{attribute 'GeneratedUsingTerminal: EK1122-0000-0018'}
{attribute addProperty BoxType "EK1122-0000-0018"}
{attribute addProperty Id "R1_A4_X2_A2_VI1_AES_D_BC_ECAT_xAES_B47A261080REX_350_IMecat_xIMecat_x_75C6CB6B170"}
{attribute addProperty CRC "967560231"}
{attribute addProperty Size "250"}
{attribute addProperty Name "R1_A4_X2_A2 (EK1122)"}
TYPE R1_A4_X2_A2_EK1122_39ABCC27 EXTENDS EK1122_1FC0878B :
STRUCT
	{attribute addProperty Name "R1_A4_X2_A2_VI1 (AES-D-BC-ECAT)"}
	{attribute addProperty PreviousPort "R1_A4_X2_A2 (EK1122) : D"}
	{attribute addProperty SyncUnit "S10"}
	R1_A4_X2_A2_VI1_AES_D_BC_ECAT_x : AES_B47A2610;
	{attribute addProperty Name "REX_350 (IMecat)"}
	{attribute addProperty PreviousPort "R1_A4_X2_A2 (EK1122) : B"}
	{attribute addProperty SyncUnit "default"}
	REX_350_IMecat_x : IMecat_x_75C6CB6B;
END_STRUCT
END_TYPE

(* stored: Version 1.2.0.0, ProductVersion 3.1.4024.11
   DUT R1_A4_X2_A2_EK1122_39ABCC27: Id {76b0b59e-c2b4-0621-0a7d-6b3058255909} *)
